% RSLogix 500 project zad1a.RSS, saved by version 8.30.00.16 %
PROJECT "P2"    % processor: Bul.1763 MicroLogix 1100 Series B %

PROGRAM FILES
  LAD 2   42 rungs

DATA FILES
  O0 OUTPUT  4 elements
  I1 INPUT  6 elements
  S2 STATUS  66 elements
  B3 BINARY  20 elements
  T4 TIMER  20 elements
  C5 COUNTER  1 elements
  R6 CONTROL  1 elements
  N7 INTEGER  1 elements
  F8 FLOAT  1 elements
  C9   1 elements

LADDER 2
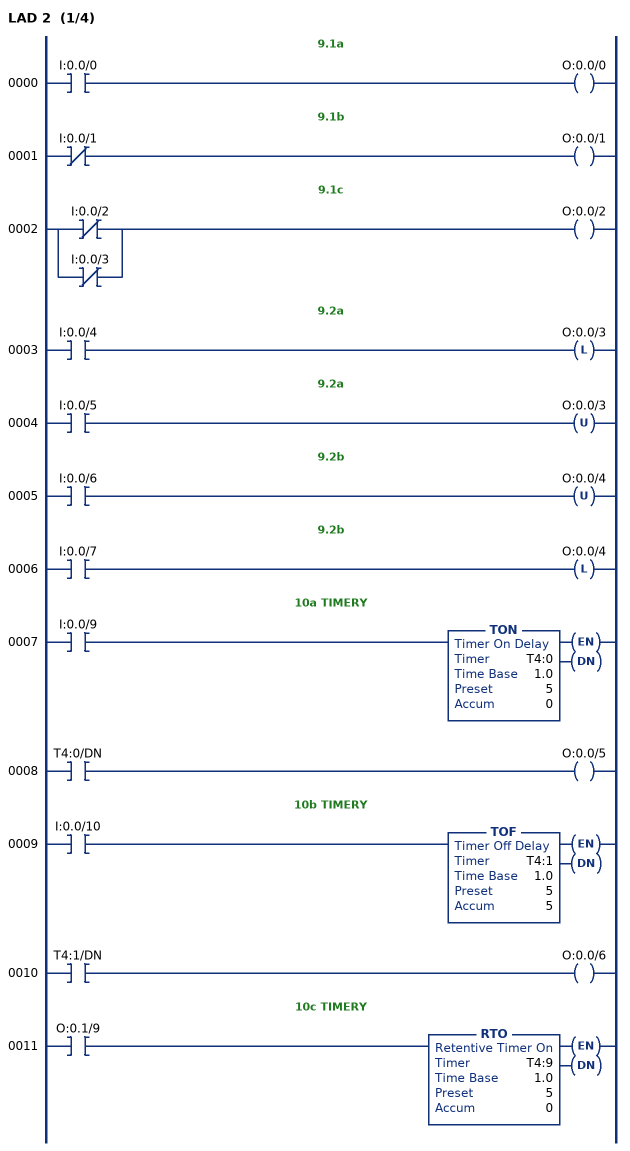
% Rung: 0 %
% TITLE: 9.1a %
SOR XIC I:0.0/0 OTE O:0.0/0 EOR
% Rung: 1 %
% TITLE: 9.1b %
SOR XIO I:0.0/1 OTE O:0.0/1 EOR
% Rung: 2 %
% TITLE: 9.1c %
SOR BST XIO I:0.0/2 NXB XIO I:0.0/3 BND OTE O:0.0/2 EOR
% Rung: 3 %
% TITLE: 9.2a %
SOR XIC I:0.0/4 OTL O:0.0/3 EOR
% Rung: 4 %
% TITLE: 9.2a %
SOR XIC I:0.0/5 OTU O:0.0/3 EOR
% Rung: 5 %
% TITLE: 9.2b %
SOR XIC I:0.0/6 OTU O:0.0/4 EOR
% Rung: 6 %
% TITLE: 9.2b %
SOR XIC I:0.0/7 OTL O:0.0/4 EOR
% Rung: 7 %
% TITLE: 10a TIMERY %
SOR XIC I:0.0/9 TON T4:0 1.0 5 0 EOR
% Rung: 8 %
SOR XIC T4:0/DN OTE O:0.0/5 EOR
% Rung: 9 %
% TITLE: 10b TIMERY %
SOR XIC I:0.0/10 TOF T4:1 1.0 5 5 EOR
% Rung: 10 %
SOR XIC T4:1/DN OTE O:0.0/6 EOR
% Rung: 11 %
% TITLE: 10c TIMERY %
SOR XIC O:0.1/9 RTO T4:9 1.0 5 0 EOR

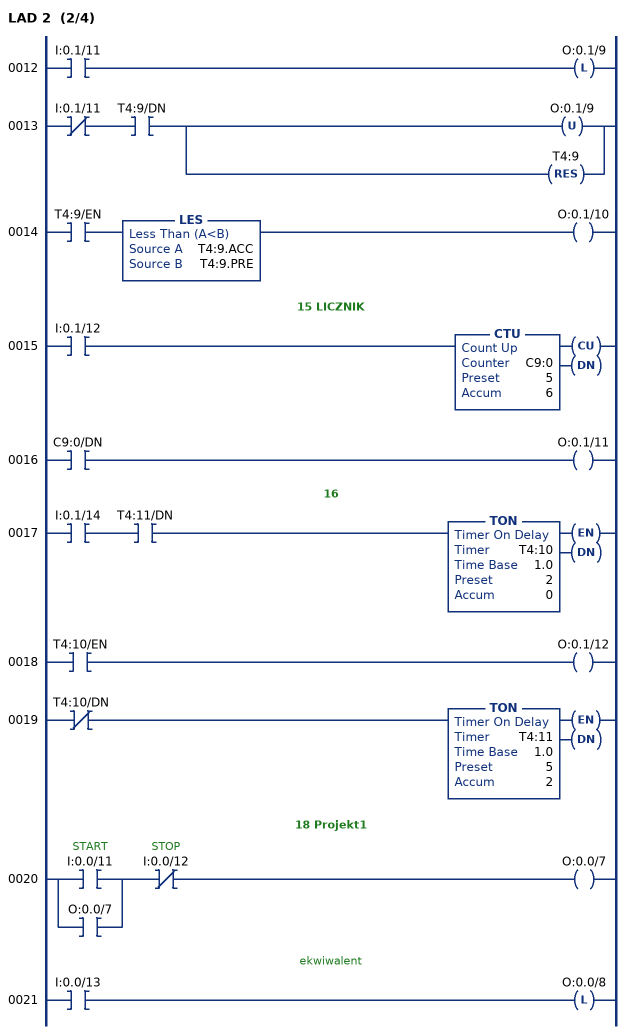
% Rung: 12 %
SOR XIC I:0.1/11 OTL O:0.1/9 EOR
% Rung: 13 %
SOR XIO I:0.1/11 XIC T4:9/DN BST OTU O:0.1/9 NXB RES T4:9 BND EOR
% Rung: 14 %
SOR XIC T4:9/EN LES T4:9.ACC T4:9.PRE OTE O:0.1/10 EOR
% Rung: 15 %
% TITLE: 15 LICZNIK %
SOR XIC I:0.1/12 CTU C9:0 5 6 EOR
% Rung: 16 %
SOR XIC C9:0/DN OTE O:0.1/11 EOR
% Rung: 17 %
% TITLE: 16 %
SOR XIC I:0.1/14 XIC T4:11/DN TON T4:10 1.0 2 0 EOR
% Rung: 18 %
SOR XIC T4:10/EN OTE O:0.1/12 EOR
% Rung: 19 %
SOR XIO T4:10/DN TON T4:11 1.0 5 2 EOR
% Rung: 20 %
% TITLE: 18 Projekt1 %
SOR BST XIC I:0.0/11 NXB XIC O:0.0/7 BND XIO I:0.0/12 OTE O:0.0/7 EOR
%   I:0.0/11  START %
%   I:0.0/12  STOP %
% Rung: 21 %
% ekwiwalent %
SOR XIC I:0.0/13 OTL O:0.0/8 EOR

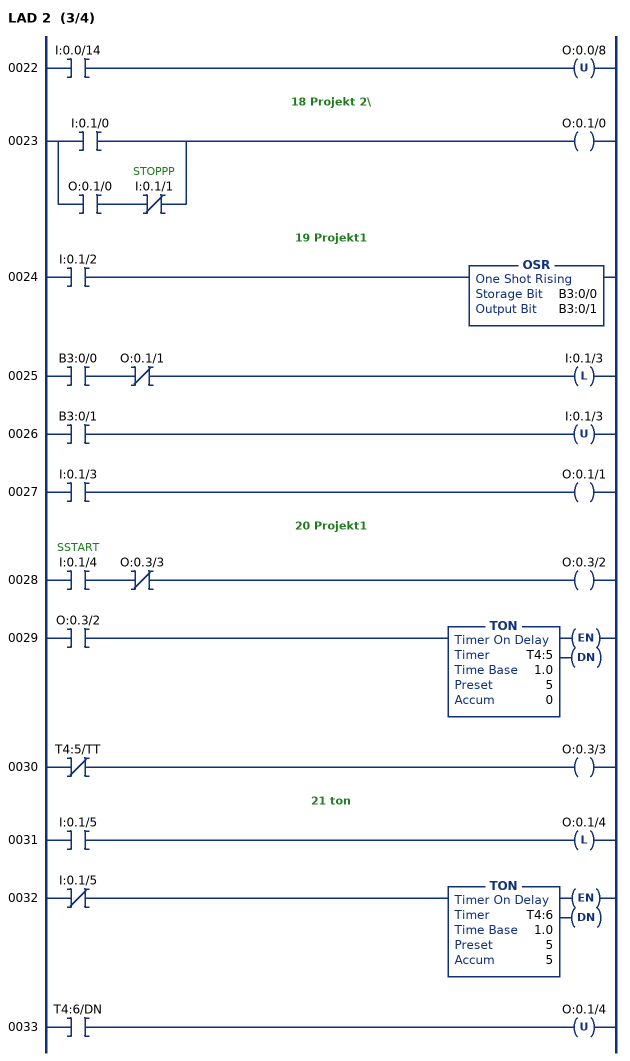
% Rung: 22 %
SOR XIC I:0.0/14 OTU O:0.0/8 EOR
% Rung: 23 %
% TITLE: 18 Projekt 2\ %
SOR BST XIC I:0.1/0 NXB XIC O:0.1/0 XIO I:0.1/1 BND OTE O:0.1/0 EOR
%   I:0.1/1  STOPPP %
% Rung: 24 %
% TITLE: 19 Projekt1 %
SOR XIC I:0.1/2 OSR B3:0/0 B3:0/1 EOR
% Rung: 25 %
SOR XIC B3:0/0 XIO O:0.1/1 OTL I:0.1/3 EOR
% Rung: 26 %
SOR XIC B3:0/1 OTU I:0.1/3 EOR
% Rung: 27 %
SOR XIC I:0.1/3 OTE O:0.1/1 EOR
% Rung: 28 %
% TITLE: 20 Projekt1 %
SOR XIC I:0.1/4 XIO O:0.3/3 OTE O:0.3/2 EOR
%   I:0.1/4  SSTART %
% Rung: 29 %
SOR XIC O:0.3/2 TON T4:5 1.0 5 0 EOR
% Rung: 30 %
SOR XIO T4:5/TT OTE O:0.3/3 EOR
% Rung: 31 %
% TITLE: 21 ton %
SOR XIC I:0.1/5 OTL O:0.1/4 EOR
% Rung: 32 %
SOR XIO I:0.1/5 TON T4:6 1.0 5 5 EOR
% Rung: 33 %
SOR XIC T4:6/DN OTU O:0.1/4 EOR

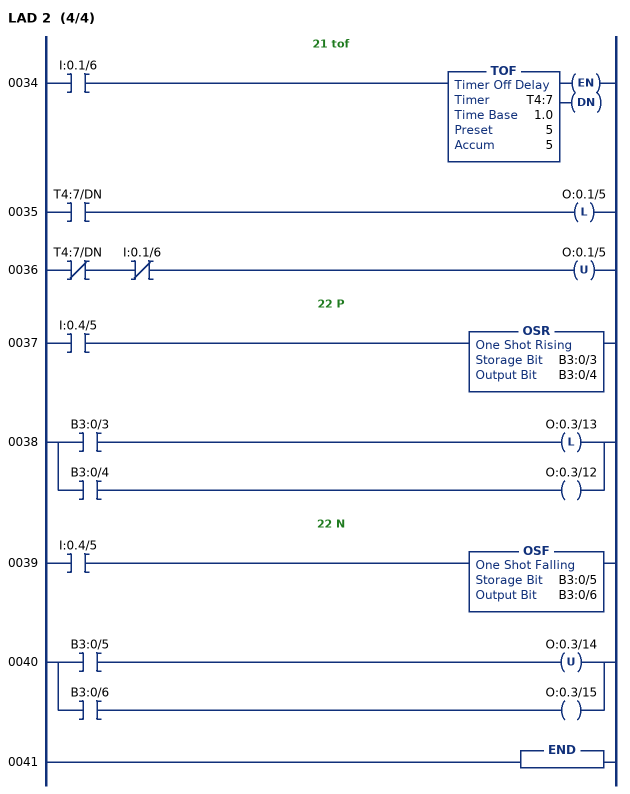
% Rung: 34 %
% TITLE: 21 tof %
SOR XIC I:0.1/6 TOF T4:7 1.0 5 5 EOR
% Rung: 35 %
SOR XIC T4:7/DN OTL O:0.1/5 EOR
% Rung: 36 %
SOR XIO T4:7/DN XIO I:0.1/6 OTU O:0.1/5 EOR
% Rung: 37 %
% TITLE: 22 P %
SOR XIC I:0.4/5 OSR B3:0/3 B3:0/4 EOR
% Rung: 38 %
SOR BST XIC B3:0/3 OTL O:0.3/13 NXB XIC B3:0/4 OTE O:0.3/12 BND EOR
% Rung: 39 %
% TITLE: 22 N %
SOR XIC I:0.4/5 OSF B3:0/5 B3:0/6 EOR
% Rung: 40 %
SOR BST XIC B3:0/5 OTU O:0.3/14 NXB XIC B3:0/6 OTE O:0.3/15 BND EOR
% Rung: 41 %
SOR END EOR

OTHER DOCUMENTED ADDRESSES
  I:1.0/1  STOP2
  I:1.1/0  START2

DATA TABLE (non-zero values as saved)
DATA T4
% .PRE .ACC %
% T4:0 % 5 0
% T4:1 % 5 5
% T4:2 % 5 0
% T4:3 % 5 0
% T4:5 % 5 0
% T4:6 % 5 5
% T4:7 % 5 5
% T4:8 % 5 0
% T4:9 % 5 0
% T4:10 % 2 0
% T4:11 % 5 2
DATA C9
% .PRE .ACC %
% C9:0 % 5 6
